// TIA Portal V19 export
DATA_BLOCK "A0304_Navetta_PERS"   // DB101
// stored: MemoryReserve 100
   VAR RETAIN
      Par : Struct
         Ax_Man : "Positioning_DOL_Machine_Par";
         Ax_Testa_Pers { ExternalAccessible := 'False'; ExternalVisible := 'False'; ExternalWritable := 'False'} : "Positioning_DOL_Machine_Pers_Data";
         Ax_Coda_Pers { ExternalAccessible := 'False'; ExternalVisible := 'False'; ExternalWritable := 'False'} : "Positioning_DOL_Machine_Pers_Data";
         Enc : Struct
            Testa : "PosFbk_RTN";
            Coda { S7_SetPoint := 'True'} : "PosFbk_RTN";
         END_STRUCT;
      END_STRUCT;
      Par_Mach : Struct
         PosPrePrelievo : LReal := -10.0;
         PosPrelievo : LReal := 0.0;
         PosDeposito : LReal := 2174.0;
         ToleranceWindow : LReal := 1.0;
      END_STRUCT;
   END_VAR
BEGIN
   Par.Ax_Man.PosTolerance := 1.0;
   Par.Ax_Man.Minus_Limit := -25.0;
   Par.Ax_Man.Plus_Limit := 2175.0;
   Par.Ax_Man.PreCutOff := 0.1;
   Par.Ax_Man.PreEndLowSpeed := 5.0;
   Par.Ax_Man.PreEndMedSpeed := 350.0;
   Par.Ax_Man.LowSpeed := 5.0;
   Par.Ax_Man.MedSpeed := 10.0;
   Par.Ax_Man.HighSpeed := 90.0;
   Par.Ax_Man.Man_Speed := 100.0;
   Par.Ax_Testa_Pers.AxisHomed := TRUE;
   Par.Ax_Coda_Pers.AxisHomed := TRUE;
   Par.Enc.Testa.Preset.Pulses := 1_965_657_700;
   Par.Enc.Testa.Preset.Units := -7.0;
   Par.Enc.Testa.Config.Resolution := -363.63935;
   Par.Enc.Coda.Preset.Pulses := -896_723_544;
   Par.Enc.Coda.Preset.Units := -7.0;
   Par.Enc.Coda.Config.Resolution := 363.63935;
END_DATA_BLOCK
